FUNCTION_BLOCK FB_DS402DriveCSP EXTENDS FB_DS402Drive
VAR_INPUT
END_VAR
VAR_OUTPUT
END_VAR
VAR
END_VAR

METHOD Abort
END_METHOD

METHOD Brake
END_METHOD

METHOD EncValue
SUPER^.EncValue();
END_METHOD

METHOD Halt : BOOL
SUPER^.Halt();
END_METHOD

{warning 'Add method implementation '}
METHOD HandleMoveRequest
END_METHOD

METHOD Home : BOOL
SUPER^.Home();
END_METHOD

METHOD Interlock
SUPER^.Interlock();
END_METHOD

METHOD Logger
END_METHOD

METHOD MotionParams
VAR_INPUT
	tRefreshDelay	: TIME;
END_VAR
SUPER^.MotionParams(tRefreshDelay);
END_METHOD

METHOD MoveAbsolute
END_METHOD

{warning 'Add method implementation '}
METHOD MoveRelative
END_METHOD

METHOD MoveVelocity
END_METHOD

METHOD Power : BOOL
SUPER^.Power();
END_METHOD

METHOD Reset : BOOL
SUPER^.Reset();
END_METHOD

METHOD SetEnables
SUPER^.SetEnables();
END_METHOD

METHOD StateMachine
SUPER^.StateMachine();
END_METHOD

END_FUNCTION_BLOCK

(* stored: Version 1.1.0.1
   POU FB_DS402DriveCSP: Id {040ef492-7146-48c0-93e4-0ac5dec2d90a}, SpecialFunc None
   Method Abort: Id {3395396f-7b35-48b5-92b0-2832ec86a6ea}
   Method Brake: Id {95fbe001-f4c7-4279-a7e0-0cb29dfca4d4}
   Method EncValue: Id {756fef2b-abd0-4ea6-a086-c6a4b4fde2ba}
   Method Halt: Id {80ebc76d-a0d6-4aeb-9553-bcbdc8add6fe}
   Method HandleMoveRequest: Id {1795147a-9aa0-450a-a77b-fe9516570119}
   Method Home: Id {879bbb12-9560-4f3a-a7e5-35aa410df12c}
   Method Interlock: Id {865c7dcc-697a-462b-bf51-9a475527ddcc}
   Method Logger: Id {14be7a94-da7c-4ae2-99d2-5034bb688728}
   Method MotionParams: Id {fe16c5bc-93e8-4071-a5cf-50df00e57f42}
   Method MoveAbsolute: Id {d147d73b-e496-4b31-b3e7-2402213adc5f}
   Method MoveRelative: Id {fe7d57b1-7f2d-4e14-a039-e0f04841a280}
   Method MoveVelocity: Id {46388d51-f1ca-4f11-8dbb-b37a8dbbec7d}
   Method Power: Id {ab76c67e-c99c-4e68-9186-e3ddad829c25}
   Method Reset: Id {3557eb7d-0afa-44ca-a231-88fb6b234dd4}
   Method SetEnables: Id {81b61160-451b-4f54-a147-9d969a192621}
   Method StateMachine: Id {ed91f64e-16df-4e75-87be-b9a709e99da3} *)
